PROGRAM MAIN
VAR
	XBoxController : FB_XBox_Controller('',1);
	
	BatteryType: XBoxControllerUtilities.E_XBox_Controller_Battery_Types;
	BatteryLevel: XBoxControllerUtilities.E_XBox_Controller_Battery_Levels;
	LeftJoystick: XBoxControllerUtilities.ST_XBox_Controller_Joystick;
END_VAR

XBoxController.Cycle();


LeftJoystick := XBoxController.P_Left_Joystick;

BatteryType := XBoxController.P_Status.Battery_Type;
BatteryLevel := XBoxController.P_Status.Battery_Level;

END_PROGRAM

(* stored: Version 1.1.0.1, ProductVersion 3.1.4024.11
   POU MAIN: Id {a9d3af89-b721-4444-bf44-98f3205fc2f1}, SpecialFunc None *)
